// TIA Portal V17 export
// export: Created 2024-08-07T21:43:53.9854891Z, ExportSetting WithDefaults, DisplayName Totally Integrated Automation Portal, DisplayVersion V17 Update 7, DisplayName TIA Portal Openness, DisplayVersion V17 Update 7, DisplayName TIA Portal Version Control Interface, DisplayVersion V17, DisplayName SINAMICS Startdrive Advanced, DisplayVersion V17 SP2, DisplayName SINAMICS Startdrive G110M, G120, G120C, G120D, G120P, G115D, DisplayVersion V17 SP2, DisplayName SINAMICS Startdrive G130, G150, S120, S150, SINAMICS MV, S210, DisplayVersion V17 SP2, DisplayName STEP 7 Professional, DisplayVersion V17 Update 7, DisplayName STEP 7 Safety, DisplayVersion V17 Update 6, DisplayName WinCC Advanced / Unified PC, DisplayVersion V17 Update 7
FUNCTION_BLOCK "CylinderFaceplate"   // FB31, LAD
{ S7_Optimized_Access := 'FALSE' }
AUTHOR : Bodorik
FAMILY : RIV
NAME : Cylinder
VERSION : 0.9
// stored: AutoNumber true, IsIECCheckEnabled false, SetENOAutomatically false, UDAEnableTagReadback false
   VAR_INPUT
      POWER_OK : Bool;
      CylinderNumber : Int;
      HMICommand : Int;
      BasicPositionCondition : Bool;
      WorkPositionCondition : Bool;
      BasicPositionSensor : Bool;
      WorkPositionSensor : Bool;
      TRIGGER : Bool;
      RESET : Bool;
      DELAY_BASIC : Time;
      DELAY_WORK : Time;
      DELAY_FREE : Time;
      ERROR_TIME : Time;
      ValveDelay : Time;
      iNoCollisionBasic : Bool;
      iNoCollisionWork : Bool;
      iNoCollisionFree : Bool;
   END_VAR
   VAR_OUTPUT
      VALVE_BASIC : Bool;
      VALVE_WORK : Bool;
      ERROR_BASIC : Bool;
      ERROR_WORK : Bool;
      HMIStatus : Int;
   END_VAR
   VAR_IN_OUT
      MOVE_BASIC : Bool;
      MOVE_WORK : Bool;
      MOVE_FREE : Bool;
      CylinderOperation : "UDT_Cylinder";
   END_VAR
   VAR DB_SPECIFIC
      "4l+Started" : Bool;
      InitCommandBP : Bool;
      InitCommandWP : Bool;
      BasicWorkStartWP : Bool;
      BasicWorkStartBP : Bool;
      work_valve : Bool;
      basic_valve : Bool;
      free_valve : Bool;
      baspos_error : TON_TIME;
      workpos_error { S7_SetPoint := 'True'} : TON_TIME;
      baspos_delay { S7_SetPoint := 'True'} : TON_TIME;
      workpos_delay { S7_SetPoint := 'True'} : TON_TIME;
      CylinderOperationOld { S7_SetPoint := 'True'} : "UDT_Cylinder";
      IEC_Timer_0_Instance { S7_SetPoint := 'True'} : TP_TIME;
   END_VAR
   VAR
      R_TRIG_Instance { S7_SetPoint := 'True'} : R_TRIG;
   END_VAR
   VAR DB_SPECIFIC
      IEC_Timer_0_Instance_1 { S7_SetPoint := 'True'} : TP_TIME;
      IEC_Timer_0_Instance_2 { S7_SetPoint := 'True'} : TP_TIME;
      IEC_Timer_0_Instance_3 { S7_SetPoint := 'True'} : TON_TIME;
      IEC_Timer_0_Instance_4 { S7_SetPoint := 'True'} : TON_TIME;
   END_VAR
   VAR_TEMP
      et : Bool;
      comm : Int;
   END_VAR
   VAR_TEMP   // added for the SCL form of the ladder/FBD networks
      _w1 : Bool;
   END_VAR
BEGIN

REGION Network 1 (SCL): check new cylinder command
   //check if basic position req movement changed
   IF #CylinderOperation.ToBp <> #CylinderOperationOld.ToBp AND #CylinderOperation.ToBp THEN
       IF #iNoCollisionBasic OR (#BasicPositionCondition AND NOT #WorkPositionCondition) THEN
           #CylinderOperation.ToFp := false;
           #CylinderOperation.ToWp := false;
       ELSE
           #CylinderOperation.ToBp := false;
       END_IF;
   END_IF;
   //check if work position req movement changed
   IF #CylinderOperation.ToWp <> #CylinderOperationOld.ToWp AND #CylinderOperation.ToWp THEN
       IF #iNoCollisionWork OR (NOT #BasicPositionCondition AND #WorkPositionCondition) THEN
           #CylinderOperation.ToFp := false;
           #CylinderOperation.ToBp := false;
       ELSE
           #CylinderOperation.ToWp := false;
       END_IF;
   END_IF;
   //check if free position req movement changed
   IF #CylinderOperation.ToFp <> #CylinderOperationOld.ToFp AND #CylinderOperation.ToFp THEN
       IF #iNoCollisionFree THEN
           #CylinderOperation.ToBp := false;
           #CylinderOperation.ToWp := false;
       ELSE
           #CylinderOperation.ToFp := false;
       END_IF;
   END_IF;
   //store actual cylinder status to old
   #CylinderOperationOld := #CylinderOperation;
END_REGION

REGION Network 2 (SCL)
   #comm := #HMICommand - #CylinderNumber;
   #CylinderOperation.ToBp := #CylinderOperation.ToBp;
   #CylinderOperation.ToWp := #CylinderOperation.ToWp;
   #MOVE_BASIC := #MOVE_BASIC;
   #MOVE_WORK := #MOVE_WORK;


   IF (#comm = 1000 AND #iNoCollisionBasic) OR #CylinderOperation.ToBp THEN
       #CylinderOperation.ToBp := true;
       #CylinderOperation.ToWp := FALSE;
       #CylinderOperation.ToFp := FALSE;
       #MOVE_BASIC := true;
       #MOVE_FREE := false;
       #MOVE_WORK := false;
   END_IF;
   IF (#comm = 2000 AND #iNoCollisionWork) OR #CylinderOperation.ToWp THEN
       #CylinderOperation.ToWp := true;
       #CylinderOperation.ToBp := FALSE;
       #CylinderOperation.ToFp := FALSE;
       #MOVE_BASIC := false;
       #MOVE_FREE := false;
       #MOVE_WORK := TRUE;
   END_IF;
   IF (#comm = 3000 AND #iNoCollisionFree) OR #CylinderOperation.ToFp THEN
       #CylinderOperation.ToFp := true;
       #CylinderOperation.ToWp := FALSE;
       #CylinderOperation.ToBp := FALSE;
       #MOVE_BASIC := FALSE;
       #MOVE_FREE := TRUE;
       #MOVE_WORK := false;
   END_IF;

   IF #ERROR_BASIC OR #ERROR_WORK THEN
       #MOVE_BASIC := 0;
       #MOVE_WORK := 0;
       #CylinderOperation.ToBp := false;
       #CylinderOperation.ToWp := false;
   END_IF;

   IF NOT #POWER_OK THEN
       #MOVE_BASIC := false;
       #MOVE_WORK := false;
       #MOVE_FREE := TRUE;
       #CylinderOperation.ToBp := false;
       #CylinderOperation.ToWp := false;
       #CylinderOperation.ToFp := TRUE;
   END_IF;
END_REGION

REGION Network 3: Start movement to basic position
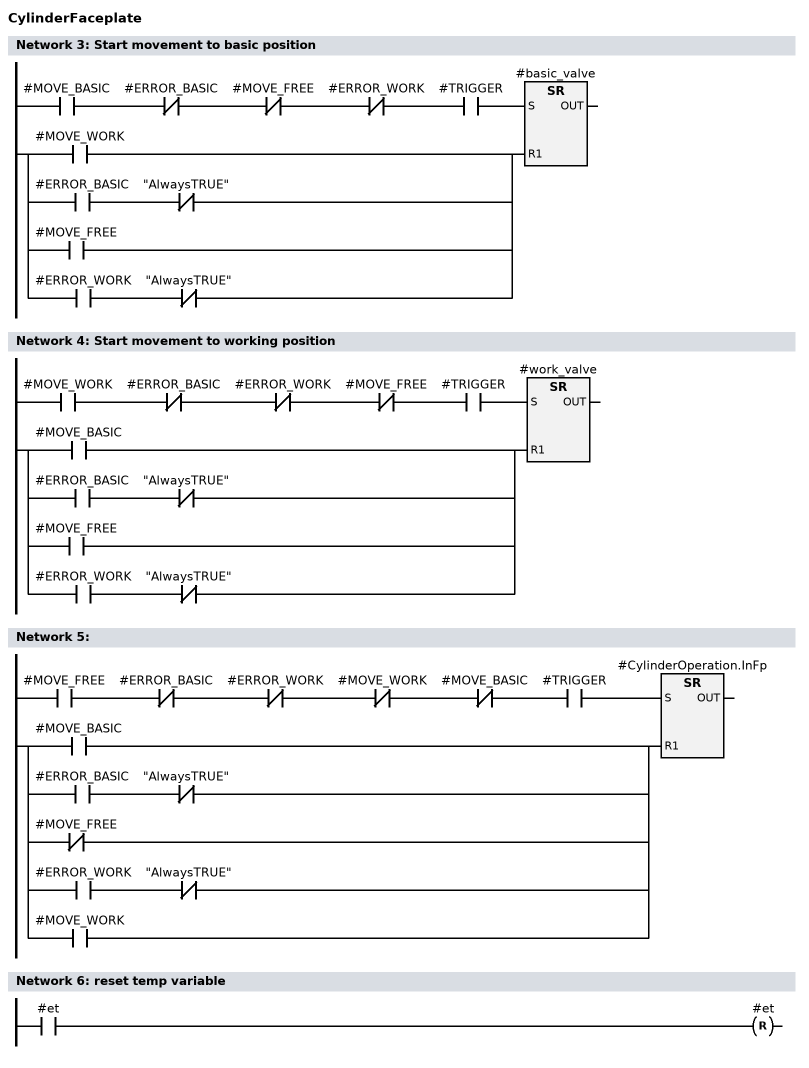
   RUNG wire#powerrail
      Contact( #MOVE_BASIC )
      I_Contact( #ERROR_BASIC )
      I_Contact( #MOVE_FREE )
      I_Contact( #ERROR_WORK )
      Contact( #TRIGGER )
      S_SR(operand := #basic_valve, r1 := wire#w1)
   END_RUNG
   RUNG wire#powerrail
      Contact( #MOVE_WORK )
   END_RUNG wire#w1
   RUNG wire#powerrail
      Contact( #ERROR_BASIC )
      I_Contact( "AlwaysTRUE" )
   END_RUNG wire#w1
   RUNG wire#powerrail
      Contact( #MOVE_FREE )
   END_RUNG wire#w1
   RUNG wire#powerrail
      Contact( #ERROR_WORK )
      I_Contact( "AlwaysTRUE" )
   END_RUNG wire#w1
   // the same network as SCL:
   IF #MOVE_BASIC AND NOT #ERROR_BASIC AND NOT #MOVE_FREE AND NOT #ERROR_WORK AND #TRIGGER THEN
       #basic_valve := TRUE;   // SR flip-flop
   END_IF;
   IF #MOVE_WORK OR (#ERROR_BASIC AND NOT "AlwaysTRUE") OR #MOVE_FREE OR (#ERROR_WORK AND NOT "AlwaysTRUE") THEN
       #basic_valve := FALSE;
   END_IF;
END_REGION

REGION Network 4: Start movement to working position
   RUNG wire#powerrail
      Contact( #MOVE_WORK )
      I_Contact( #ERROR_BASIC )
      I_Contact( #ERROR_WORK )
      I_Contact( #MOVE_FREE )
      Contact( #TRIGGER )
      S_SR(operand := #work_valve, r1 := wire#w1)
   END_RUNG
   RUNG wire#powerrail
      Contact( #MOVE_BASIC )
   END_RUNG wire#w1
   RUNG wire#powerrail
      Contact( #ERROR_BASIC )
      I_Contact( "AlwaysTRUE" )
   END_RUNG wire#w1
   RUNG wire#powerrail
      Contact( #MOVE_FREE )
   END_RUNG wire#w1
   RUNG wire#powerrail
      Contact( #ERROR_WORK )
      I_Contact( "AlwaysTRUE" )
   END_RUNG wire#w1
   // the same network as SCL:
   IF #MOVE_WORK AND NOT #ERROR_BASIC AND NOT #ERROR_WORK AND NOT #MOVE_FREE AND #TRIGGER THEN
       #work_valve := TRUE;   // SR flip-flop
   END_IF;
   IF #MOVE_BASIC OR (#ERROR_BASIC AND NOT "AlwaysTRUE") OR #MOVE_FREE OR (#ERROR_WORK AND NOT "AlwaysTRUE") THEN
       #work_valve := FALSE;
   END_IF;
END_REGION

REGION Network 5
   RUNG wire#powerrail
      Contact( #MOVE_FREE )
      I_Contact( #ERROR_BASIC )
      I_Contact( #ERROR_WORK )
      I_Contact( #MOVE_WORK )
      I_Contact( #MOVE_BASIC )
      Contact( #TRIGGER )
      S_SR(operand := #CylinderOperation.InFp, r1 := wire#w1)
   END_RUNG
   RUNG wire#powerrail
      Contact( #MOVE_BASIC )
   END_RUNG wire#w1
   RUNG wire#powerrail
      Contact( #ERROR_BASIC )
      I_Contact( "AlwaysTRUE" )
   END_RUNG wire#w1
   RUNG wire#powerrail
      I_Contact( #MOVE_FREE )
   END_RUNG wire#w1
   RUNG wire#powerrail
      Contact( #ERROR_WORK )
      I_Contact( "AlwaysTRUE" )
   END_RUNG wire#w1
   RUNG wire#powerrail
      Contact( #MOVE_WORK )
   END_RUNG wire#w1
   // the same network as SCL:
   IF #MOVE_FREE AND NOT #ERROR_BASIC AND NOT #ERROR_WORK AND NOT #MOVE_WORK AND NOT #MOVE_BASIC AND #TRIGGER THEN
       #CylinderOperation.InFp := TRUE;   // SR flip-flop
   END_IF;
   IF #MOVE_BASIC OR (#ERROR_BASIC AND NOT "AlwaysTRUE") OR NOT #MOVE_FREE OR (#ERROR_WORK AND NOT "AlwaysTRUE") OR #MOVE_WORK THEN
       #CylinderOperation.InFp := FALSE;
   END_IF;
END_REGION

REGION Network 6: reset temp variable
   RUNG wire#powerrail
      Contact( #et )
      R_Coil( #et )
   END_RUNG
   // the same network as SCL:
   IF #et THEN #et := FALSE; END_IF;
END_REGION

REGION Network 7 (FBD): Error movement to basic position
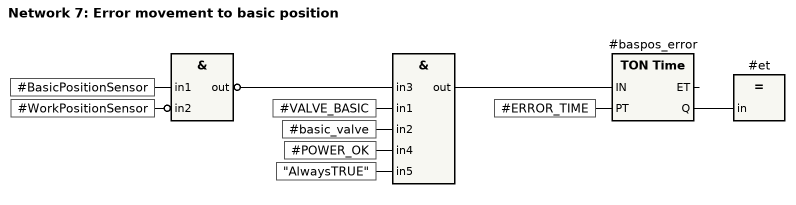
   #baspos_error(IN := NOT (#BasicPositionSensor AND NOT #WorkPositionSensor) AND #VALVE_BASIC AND #basic_valve AND #POWER_OK AND "AlwaysTRUE",   // TON
                 PT := #ERROR_TIME);
   #et := #baspos_error.Q;
END_REGION

REGION Network 8: Set basic position error
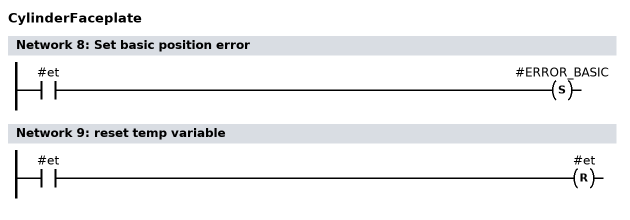
   RUNG wire#powerrail
      Contact( #et )
      S_Coil( #ERROR_BASIC )
   END_RUNG
   // the same network as SCL:
   IF #et THEN #ERROR_BASIC := TRUE; END_IF;
END_REGION

REGION Network 9: reset temp variable
   RUNG wire#powerrail
      Contact( #et )
      R_Coil( #et )
   END_RUNG
   // the same network as SCL:
   IF #et THEN #et := FALSE; END_IF;
END_REGION

REGION Network 10 (FBD): Error movement to working position
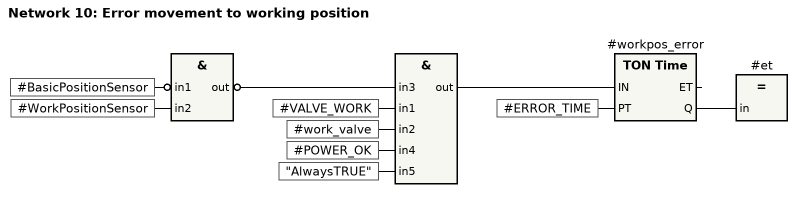
   #workpos_error(IN := NOT (NOT #BasicPositionSensor AND #WorkPositionSensor) AND #VALVE_WORK AND #work_valve AND #POWER_OK AND "AlwaysTRUE",   // TON
                  PT := #ERROR_TIME);
   #et := #workpos_error.Q;
END_REGION

REGION Network 11: Set working position error
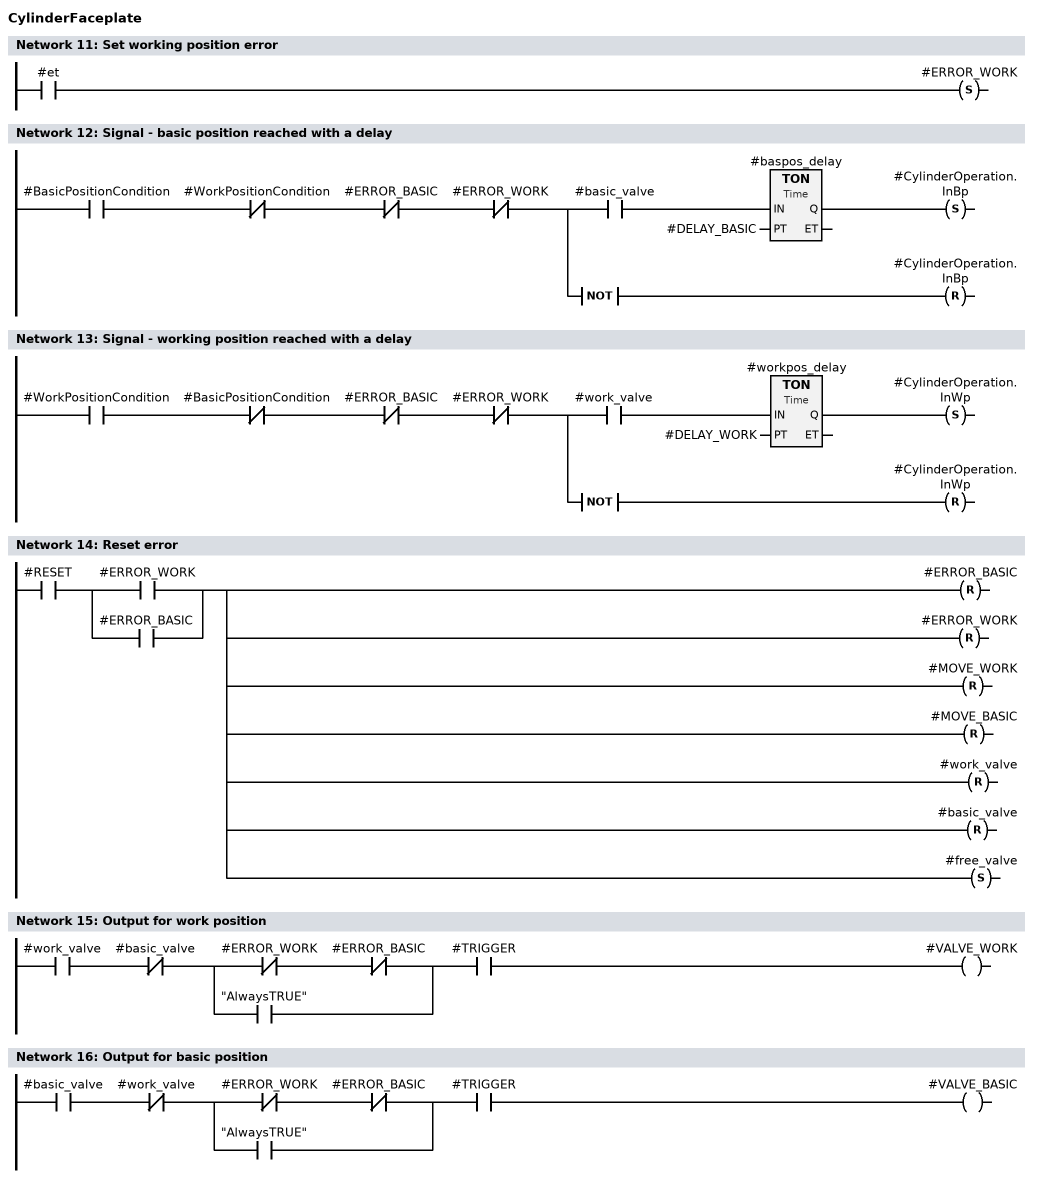
   RUNG wire#powerrail
      Contact( #et )
      S_Coil( #ERROR_WORK )
   END_RUNG
   // the same network as SCL:
   IF #et THEN #ERROR_WORK := TRUE; END_IF;
END_REGION

REGION Network 12: Signal - basic position reached with a delay
   RUNG wire#powerrail
      Contact( #BasicPositionCondition )
      I_Contact( #WorkPositionCondition )
      I_Contact( #ERROR_BASIC )
      I_Contact( #ERROR_WORK )
      wire#w1
      Contact( #basic_valve )
      { S7_Templates := "time_type := Time" } #baspos_delay.TON(pt := #DELAY_BASIC, et =>)
      S_Coil( #CylinderOperation.InBp )
   END_RUNG
   RUNG wire#w1
      Not()
      R_Coil( #CylinderOperation.InBp )
   END_RUNG
   // the same network as SCL:
   #_w1 := #BasicPositionCondition AND NOT #WorkPositionCondition AND NOT #ERROR_BASIC AND NOT #ERROR_WORK;
   #baspos_delay(IN := #_w1 AND #basic_valve, PT := #DELAY_BASIC);   // TON
   IF #baspos_delay.Q THEN #CylinderOperation.InBp := TRUE; END_IF;
   IF NOT #_w1 THEN #CylinderOperation.InBp := FALSE; END_IF;
END_REGION

REGION Network 13: Signal - working position reached with a delay
   RUNG wire#powerrail
      Contact( #WorkPositionCondition )
      I_Contact( #BasicPositionCondition )
      I_Contact( #ERROR_BASIC )
      I_Contact( #ERROR_WORK )
      wire#w1
      Contact( #work_valve )
      { S7_Templates := "time_type := Time" } #workpos_delay.TON(pt := #DELAY_WORK, et =>)
      S_Coil( #CylinderOperation.InWp )
   END_RUNG
   RUNG wire#w1
      Not()
      R_Coil( #CylinderOperation.InWp )
   END_RUNG
   // the same network as SCL:
   #_w1 := #WorkPositionCondition AND NOT #BasicPositionCondition AND NOT #ERROR_BASIC AND NOT #ERROR_WORK;
   #workpos_delay(IN := #_w1 AND #work_valve, PT := #DELAY_WORK);   // TON
   IF #workpos_delay.Q THEN #CylinderOperation.InWp := TRUE; END_IF;
   IF NOT #_w1 THEN #CylinderOperation.InWp := FALSE; END_IF;
END_REGION

REGION Network 14: Reset error
   RUNG wire#powerrail
      Contact( #RESET )
      wire#w1
      Contact( #ERROR_WORK )
      wire#w2
      R_Coil( #ERROR_BASIC )
   END_RUNG
   RUNG wire#w1
      Contact( #ERROR_BASIC )
   END_RUNG wire#w2
   RUNG wire#w2
      R_Coil( #ERROR_WORK )
   END_RUNG
   RUNG wire#w2
      R_Coil( #MOVE_WORK )
   END_RUNG
   RUNG wire#w2
      R_Coil( #MOVE_BASIC )
   END_RUNG
   RUNG wire#w2
      R_Coil( #work_valve )
   END_RUNG
   RUNG wire#w2
      R_Coil( #basic_valve )
   END_RUNG
   RUNG wire#w2
      S_Coil( #free_valve )
   END_RUNG
   // the same network as SCL:
   #_w1 := #RESET AND (#ERROR_WORK OR #ERROR_BASIC);
   IF #_w1 THEN
       #ERROR_BASIC := FALSE;
       #ERROR_WORK := FALSE;
       #MOVE_WORK := FALSE;
       #MOVE_BASIC := FALSE;
       #work_valve := FALSE;
       #basic_valve := FALSE;
       #free_valve := TRUE;
   END_IF;
END_REGION

REGION Network 15: Output for work position
   RUNG wire#powerrail
      Contact( #work_valve )
      I_Contact( #basic_valve )
      wire#w1
      I_Contact( #ERROR_WORK )
      I_Contact( #ERROR_BASIC )
      wire#w2
      Contact( #TRIGGER )
      Coil( #VALVE_WORK )
   END_RUNG
   RUNG wire#w1
      Contact( "AlwaysTRUE" )
   END_RUNG wire#w2
   // the same network as SCL:
   #VALVE_WORK := #work_valve AND NOT #basic_valve AND ((NOT #ERROR_WORK AND NOT #ERROR_BASIC) OR "AlwaysTRUE") AND #TRIGGER;
END_REGION

REGION Network 16: Output for basic position
   RUNG wire#powerrail
      Contact( #basic_valve )
      I_Contact( #work_valve )
      wire#w1
      I_Contact( #ERROR_WORK )
      I_Contact( #ERROR_BASIC )
      wire#w2
      Contact( #TRIGGER )
      Coil( #VALVE_BASIC )
   END_RUNG
   RUNG wire#w1
      Contact( "AlwaysTRUE" )
   END_RUNG wire#w2
   // the same network as SCL:
   #VALVE_BASIC := #basic_valve AND NOT #work_valve AND ((NOT #ERROR_WORK AND NOT #ERROR_BASIC) OR "AlwaysTRUE") AND #TRIGGER;
END_REGION

REGION Network 17 (SCL): Count status integer to HMI
   #comm := 0;
   IF #BasicPositionSensor THEN
       #comm := #comm + w#16#01;
   END_IF;

   IF #WorkPositionSensor THEN
       #comm := #comm + w#16#02;
   END_IF;

   IF #ERROR_BASIC THEN
       #comm := #comm + w#16#0040;
   END_IF;

   IF #ERROR_WORK THEN
       #comm := #comm + w#16#0080;
   END_IF;

   IF #VALVE_BASIC THEN
       #comm := #comm + w#16#0100;
   END_IF;
   IF #VALVE_WORK THEN
       #comm := #comm + w#16#0200;
   END_IF;

   IF NOT #iNoCollisionBasic THEN
       #comm := #comm + w#16#08;
   END_IF;

   IF NOT #iNoCollisionWork THEN
       #comm := #comm + w#16#10;
   END_IF;

   IF NOT #iNoCollisionFree THEN
       #comm := #comm + w#16#20;
   END_IF;

   #HMIStatus := #comm;
END_REGION
END_FUNCTION_BLOCK
